PROGRAM Turret_Manager
VAR
	Turret_Offset: LREAL;	
	ExtraSensorInput: TAxSensorModule; // compressed FUN for exteriour sensor inputs. temp, edge, jog stops
	SpecialOperations: TAxSpecialOperationModule; //compressed FUN for the special operation commands. 
	AxisCoupleIN: TAxCoupleModule; //connects to the AX_Couple_out of the manager from the next axis. NOT MASTER/SLAVE
	ErrorWordArray: WORD; //build a array of words that act as a cluster of error watching variables. each step in array will be one axis. differant values of the word for each axis mean a differant error. 
	JogStop: LREAL := 1E100 ; // a stopping point using the jog system to signify it is in the right spot. Need to have the LimitPosJOG adjusted after to compensate for the next space.
	DriveCMD_1: DriveCMDShortCUT; //extra system for the FB to make it easy to read.
	ASPshortCut_1: ASPshortCUT;  // same as above
	Achs_Return_Turret: TAxReturn;
END_VAR

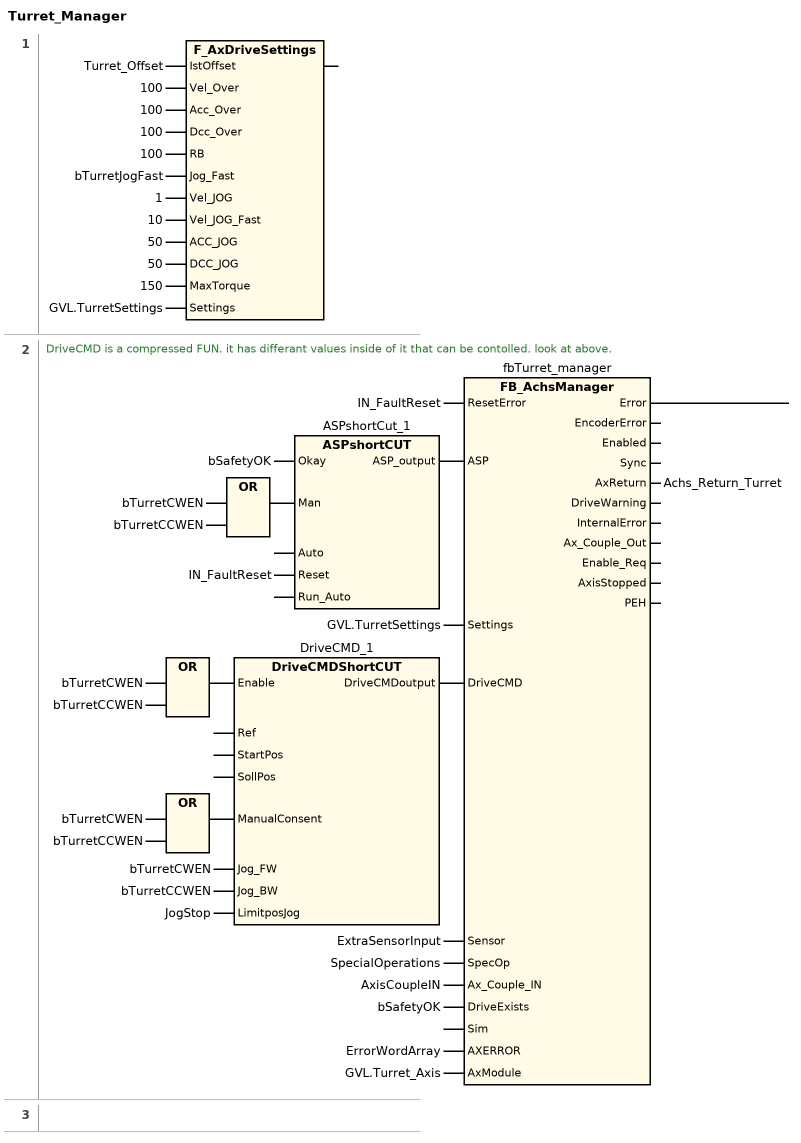
// NETWORK 1
F_AxDriveSettings(IstOffset := Turret_Offset, Vel_Over := 100, Acc_Over := 100, Dcc_Over := 100, RB := 100, Jog_Fast := bTurretJogFast, Vel_JOG := 1, Vel_JOG_Fast := 10, ACC_JOG := 50, DCC_JOG := 50, MaxTorque := 150, Settings := GVL.TurretSettings);

// NETWORK 2
// DriveCMD is a compressed FUN. it has differant values inside of it that can be contolled. look at above.
ASPshortCut_1(Okay := bSafetyOK, Man := bTurretCWEN OR bTurretCCWEN, Reset := IN_FaultReset); // ASPshortCUT
DriveCMD_1(
    Enable := bTurretCWEN OR bTurretCCWEN,
    ManualConsent := bTurretCWEN OR bTurretCCWEN,
    Jog_FW := bTurretCWEN,
    Jog_BW := bTurretCCWEN,
    LimitposJog := JogStop); // DriveCMDShortCUT
fbTurret_manager(
    ResetError := IN_FaultReset,
    ASP := ASPshortCut_1.ASP_output,
    Settings := GVL.TurretSettings,
    DriveCMD := DriveCMD_1.DriveCMDoutput,
    Sensor := ExtraSensorInput,
    SpecOp := SpecialOperations,
    Ax_Couple_IN := AxisCoupleIN,
    DriveExists := bSafetyOK,
    AXERROR := ErrorWordArray,
    AxModule := GVL.Turret_Axis,
    AxReturn => Achs_Return_Turret); // FB_AchsManager

// NETWORK 3

END_PROGRAM

(* stored: Version 1.1.0.1, ProductVersion 3.1.4024.15
   POU Turret_Manager: Id {9c872562-ea40-4b5a-ad22-d9728eb92fec}, SpecialFunc None *)
